INTERFACE I_Station

METHOD Clear : BOOL
VAR_INPUT
END_VAR
END_METHOD

METHOD Cycle : BOOL
VAR_INPUT
END_VAR
END_METHOD

METHOD Init : BOOL
END_METHOD

PROPERTY P_bInitDone : BOOL
GET
END_GET
END_PROPERTY

PROPERTY P_eProcessMode : E_ProcessMode
GET
END_GET
SET
END_SET
END_PROPERTY

PROPERTY P_List_Station : I_List
GET
END_GET
END_PROPERTY

PROPERTY P_List_Switch_Input_E : I_List
GET
END_GET
END_PROPERTY

PROPERTY P_List_Switch_Input_N : I_List
GET
END_GET
END_PROPERTY

PROPERTY P_List_Switch_Input_S : I_List
GET
END_GET
END_PROPERTY

PROPERTY P_List_Switch_Input_W : I_List
GET
END_GET
END_PROPERTY

PROPERTY P_nErrorCode : UDINT
GET
END_GET
END_PROPERTY

PROPERTY P_Position : ST_StationPosition
GET
END_GET
END_PROPERTY

PROPERTY P_ProcessClearance : DINT
GET
END_GET
END_PROPERTY

PROPERTY P_ProcessRequest : UDINT
GET
END_GET
SET
END_SET
END_PROPERTY

PROPERTY P_ProcessState : UDINT
GET
END_GET
END_PROPERTY

PROPERTY P_StationTaskList : array[1..200] of UDINT
GET
END_GET
SET
END_SET
END_PROPERTY

METHOD Process : BOOL
END_METHOD

END_INTERFACE

(* stored: Version 1.1.0.1
   Itf I_Station: Id {b7c4e6a8-f5ef-4a85-9c38-d9540037c3bc}
   Method Clear: Id {91060713-2ed2-42e7-bb37-b1107a5e6c65}
   Method Cycle: Id {a75c557b-6c9f-4cc4-b97e-1ec3d822b4a0}
   Method Init: Id {aa78eb2b-d070-4fbe-860c-b25f4b451a5c}
   Property P_bInitDone: Id {03b99a46-2131-4358-8ee2-78b639c921ea}
   Get Get: Id {64e1cb95-c985-4317-932c-fc2ebef47049}
   Property P_eProcessMode: Id {cf92a65d-6956-4c06-b3e5-f40f99fa0b52}
   Get Get: Id {18435ddd-988d-4a00-9493-fb9ff91da3ba}
   Set Set: Id {194ceb23-b84b-42b0-a605-118fc0dd5a15}
   Property P_List_Station: Id {43d2d18b-96a9-4239-9a98-df84662159be}
   Get Get: Id {9bacb839-5958-41a2-a26a-da703e2364b0}
   Property P_List_Switch_Input_E: Id {44f932a5-9164-43b5-949c-4677d15cfc6a}
   Get Get: Id {5cd63f5e-8936-4d99-b194-24c8a9c3d0a8}
   Property P_List_Switch_Input_N: Id {5a07aa47-ac5a-4c4e-8118-33b525b47208}
   Get Get: Id {e2b5108a-3276-41d0-98d4-107fe26a24c6}
   Property P_List_Switch_Input_S: Id {c14ac153-0198-4c9d-855a-bcb9d1602995}
   Get Get: Id {dcbb7747-a243-4be6-b0ae-9d984db1ac06}
   Property P_List_Switch_Input_W: Id {b3f7a703-dc33-4235-bf3d-15450c9a5650}
   Get Get: Id {98b07056-4df2-41b8-9ab8-695dd8e8fc41}
   Property P_nErrorCode: Id {ea1b2323-87e9-4702-bc65-6c2b9287f539}
   Get Get: Id {424a2654-461c-449e-9b25-ce4fe72a35e7}
   Property P_Position: Id {79b899ad-e234-49d0-8fda-9307f846f068}
   Get Get: Id {ae624e8b-fed0-4343-8088-ad6ec5760740}
   Property P_ProcessClearance: Id {8f7a4b8e-d3f3-416c-adfd-f2dd9b066afd}
   Get Get: Id {94f45565-a3e4-4d3f-89d5-ec03df4554f5}
   Property P_ProcessRequest: Id {fb31ea4d-dc37-4288-b3db-b21cbadbf4c9}
   Get Get: Id {b9dd3435-4073-4350-95ed-94e96100e900}
   Set Set: Id {1f274383-a710-4883-8c62-996464c47fcf}
   Property P_ProcessState: Id {061557d0-be34-4687-a7da-28e4efc8acab}
   Get Get: Id {815a71fc-44b4-40b9-af1e-359ba452e982}
   Property P_StationTaskList: Id {80f327e1-32e7-474b-a9a8-9774803aafcd}
   Get Get: Id {2f8e5f76-9d03-4673-8517-469f181b3d34}
   Set Set: Id {47a26ff0-59b3-43fc-948e-d2182d0d497d}
   Method Process: Id {4748aef3-ba14-429a-a8b6-29679e986082} *)
